// TIA Portal V15.1 export
// export: Created 2024-05-17T05:38:54.5998709Z, ExportSetting WithDefaults, DisplayName Totally Integrated Automation Portal, DisplayVersion V15.1 Update 5, DisplayName TIA Portal Openness, DisplayVersion V15.1 Update 5, DisplayName SINAMICS Startdrive Advanced, DisplayVersion V15.1, DisplayName G130, G150, S120, S150, SINAMICS MV, S210, DisplayVersion V15.1, DisplayName G110M, G120, G120C, G120D, G120P, DisplayVersion V15.1, DisplayName STEP 7 Professional, DisplayVersion V15.1 Update 5, DisplayName STEP 7 Safety, DisplayVersion V15.1, DisplayName WinCC Professional, DisplayVersion V15.1 Update 5, DisplayName SIMATIC Visualization Architect, DisplayVersion V15.1
FUNCTION "209220ZS01PNIODiag" : Void   // FC374, FBD
TITLE = 209220ZS01PNIODiag
{ S7_Optimized_Access := 'FALSE' }
AUTHOR : JS
NAME : Mot001
VERSION : 0.1
// stored: AutoNumber false, IsIECCheckEnabled false, SetENOAutomatically False, UDAEnableTagReadback false
   VAR_OUTPUT
      O_AlarmA : Bool;   // Alarm A
      O_AlarmB : Bool;   // Alarm B
      O_AlarmC : Bool;   // Alarm C
      O_AlarmD : Bool;   // Alarm D
      O_AlarmABCondition : Bool;   // Alarms resetable
      H_IAnim : Word;   // Animation bits to Icon in WinCC
   END_VAR
   VAR_TEMP   // added for the SCL form of the ladder/FBD networks
      _w1 : Bool;
   END_VAR
BEGIN

REGION Network 1: **** --------------------- ET200sp I/O --------------------- ****
END_REGION

REGION Network 2: **** 3 - Communication - Devices **** 209220AS10-JW50 - ET200sp I/O - Busnode 220AS10 - node 50
   // Profinet device don't exist - ET200sp I/O - Busnode 220AS10 - node 50
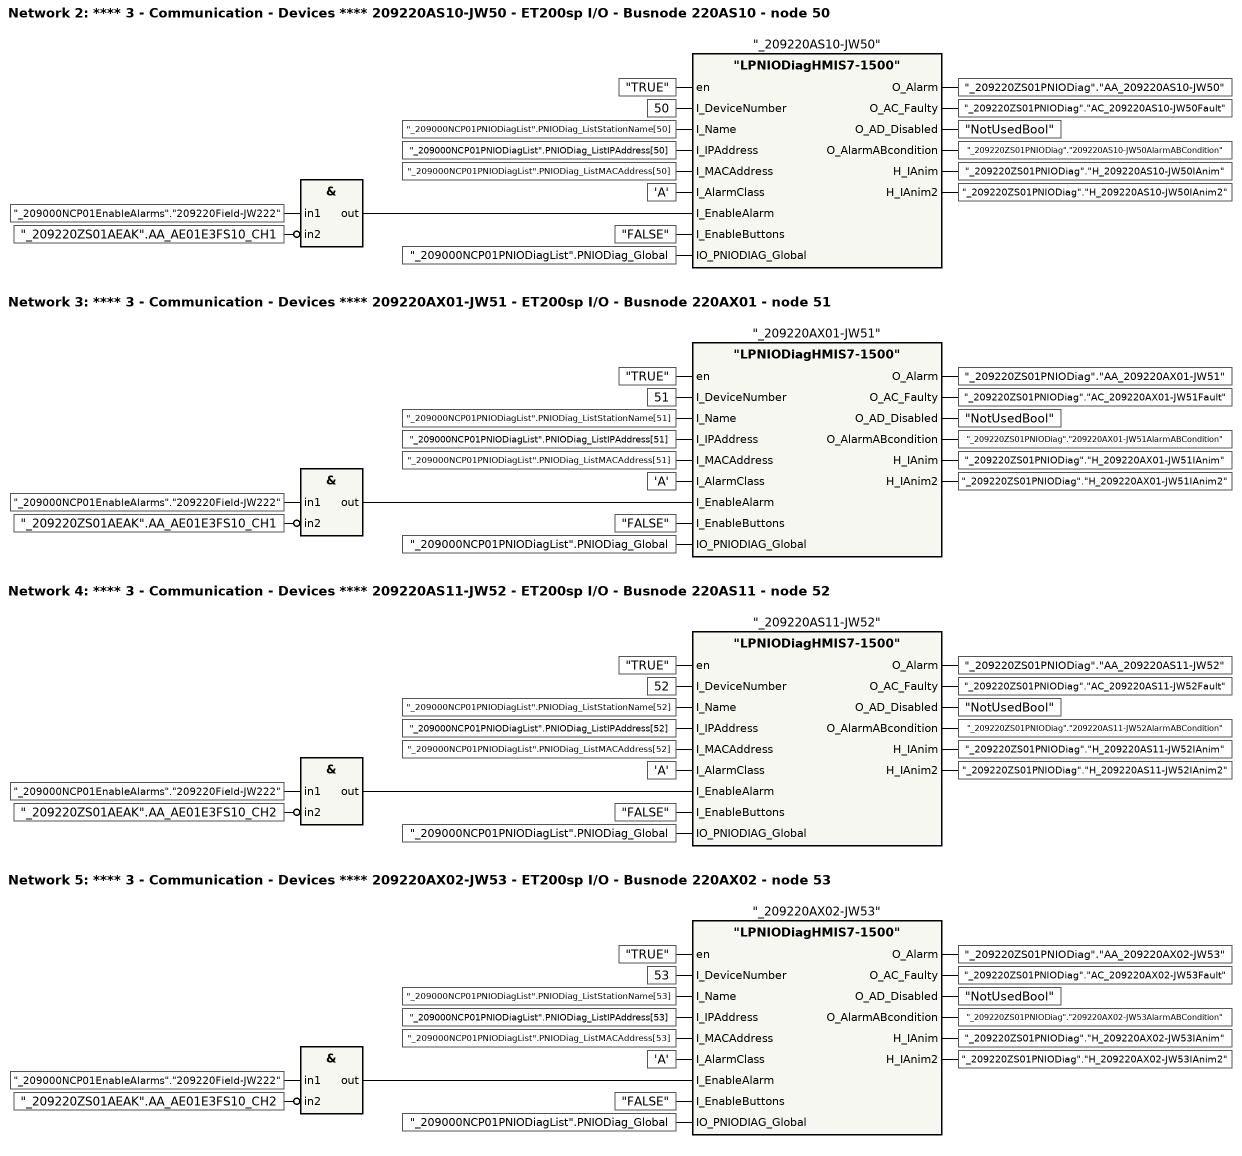
   IF "TRUE" THEN
       "_209220AS10-JW50"(I_DeviceNumber := 50,   // "LPNIODiagHMIS7-1500"
                          I_Name := "_209000NCP01PNIODiagList".PNIODiag_ListStationName[50],
                          I_IPAddress := "_209000NCP01PNIODiagList".PNIODiag_ListIPAddress[50],
                          I_MACAddress := "_209000NCP01PNIODiagList".PNIODiag_ListMACAddress[50],
                          I_AlarmClass := 'A',
                          I_EnableAlarm := "_209000NCP01EnableAlarms"."209220Field-JW222" AND NOT "_209220ZS01AEAK".AA_AE01E3FS10_CH1,
                          I_EnableButtons := "FALSE",
                          IO_PNIODIAG_Global := "_209000NCP01PNIODiagList".PNIODiag_Global,
                          O_Alarm => "_209220ZS01PNIODiag"."AA_209220AS10-JW50",
                          O_AC_Faulty => "_209220ZS01PNIODiag"."AC_209220AS10-JW50Fault",
                          O_AD_Disabled => "NotUsedBool",
                          O_AlarmABcondition => "_209220ZS01PNIODiag"."209220AS10-JW50AlarmABCondition",
                          H_IAnim => "_209220ZS01PNIODiag"."H_209220AS10-JW50IAnim",
                          H_IAnim2 => "_209220ZS01PNIODiag"."H_209220AS10-JW50IAnim2");
   END_IF;
END_REGION

REGION Network 3: **** 3 - Communication - Devices **** 209220AX01-JW51 - ET200sp I/O - Busnode 220AX01 - node 51
   // Profinet device don't exist - ET200sp I/O - Busnode 220AX01 - node 51
   IF "TRUE" THEN
       "_209220AX01-JW51"(I_DeviceNumber := 51,   // "LPNIODiagHMIS7-1500"
                          I_Name := "_209000NCP01PNIODiagList".PNIODiag_ListStationName[51],
                          I_IPAddress := "_209000NCP01PNIODiagList".PNIODiag_ListIPAddress[51],
                          I_MACAddress := "_209000NCP01PNIODiagList".PNIODiag_ListMACAddress[51],
                          I_AlarmClass := 'A',
                          I_EnableAlarm := "_209000NCP01EnableAlarms"."209220Field-JW222" AND NOT "_209220ZS01AEAK".AA_AE01E3FS10_CH1,
                          I_EnableButtons := "FALSE",
                          IO_PNIODIAG_Global := "_209000NCP01PNIODiagList".PNIODiag_Global,
                          O_Alarm => "_209220ZS01PNIODiag"."AA_209220AX01-JW51",
                          O_AC_Faulty => "_209220ZS01PNIODiag"."AC_209220AX01-JW51Fault",
                          O_AD_Disabled => "NotUsedBool",
                          O_AlarmABcondition => "_209220ZS01PNIODiag"."209220AX01-JW51AlarmABCondition",
                          H_IAnim => "_209220ZS01PNIODiag"."H_209220AX01-JW51IAnim",
                          H_IAnim2 => "_209220ZS01PNIODiag"."H_209220AX01-JW51IAnim2");
   END_IF;
END_REGION

REGION Network 4: **** 3 - Communication - Devices **** 209220AS11-JW52 - ET200sp I/O - Busnode 220AS11 - node 52
   // Profinet device don't exist - ET200sp I/O - Busnode 220AS11 - node 52
   IF "TRUE" THEN
       "_209220AS11-JW52"(I_DeviceNumber := 52,   // "LPNIODiagHMIS7-1500"
                          I_Name := "_209000NCP01PNIODiagList".PNIODiag_ListStationName[52],
                          I_IPAddress := "_209000NCP01PNIODiagList".PNIODiag_ListIPAddress[52],
                          I_MACAddress := "_209000NCP01PNIODiagList".PNIODiag_ListMACAddress[52],
                          I_AlarmClass := 'A',
                          I_EnableAlarm := "_209000NCP01EnableAlarms"."209220Field-JW222" AND NOT "_209220ZS01AEAK".AA_AE01E3FS10_CH2,
                          I_EnableButtons := "FALSE",
                          IO_PNIODIAG_Global := "_209000NCP01PNIODiagList".PNIODiag_Global,
                          O_Alarm => "_209220ZS01PNIODiag"."AA_209220AS11-JW52",
                          O_AC_Faulty => "_209220ZS01PNIODiag"."AC_209220AS11-JW52Fault",
                          O_AD_Disabled => "NotUsedBool",
                          O_AlarmABcondition => "_209220ZS01PNIODiag"."209220AS11-JW52AlarmABCondition",
                          H_IAnim => "_209220ZS01PNIODiag"."H_209220AS11-JW52IAnim",
                          H_IAnim2 => "_209220ZS01PNIODiag"."H_209220AS11-JW52IAnim2");
   END_IF;
END_REGION

REGION Network 5: **** 3 - Communication - Devices **** 209220AX02-JW53 - ET200sp I/O - Busnode 220AX02 - node 53
   // Profinet device don't exist - ET200sp I/O - Busnode 220AX02 - node 53
   IF "TRUE" THEN
       "_209220AX02-JW53"(I_DeviceNumber := 53,   // "LPNIODiagHMIS7-1500"
                          I_Name := "_209000NCP01PNIODiagList".PNIODiag_ListStationName[53],
                          I_IPAddress := "_209000NCP01PNIODiagList".PNIODiag_ListIPAddress[53],
                          I_MACAddress := "_209000NCP01PNIODiagList".PNIODiag_ListMACAddress[53],
                          I_AlarmClass := 'A',
                          I_EnableAlarm := "_209000NCP01EnableAlarms"."209220Field-JW222" AND NOT "_209220ZS01AEAK".AA_AE01E3FS10_CH2,
                          I_EnableButtons := "FALSE",
                          IO_PNIODIAG_Global := "_209000NCP01PNIODiagList".PNIODiag_Global,
                          O_Alarm => "_209220ZS01PNIODiag"."AA_209220AX02-JW53",
                          O_AC_Faulty => "_209220ZS01PNIODiag"."AC_209220AX02-JW53Fault",
                          O_AD_Disabled => "NotUsedBool",
                          O_AlarmABcondition => "_209220ZS01PNIODiag"."209220AX02-JW53AlarmABCondition",
                          H_IAnim => "_209220ZS01PNIODiag"."H_209220AX02-JW53IAnim",
                          H_IAnim2 => "_209220ZS01PNIODiag"."H_209220AX02-JW53IAnim2");
   END_IF;
END_REGION

REGION Network 6: **** 3 - Communication - Devices **** 209220AS20-JW58 - ET200sp I/O - Busnode 220AS20 - node 58
   // Profinet device don't exist - ET200sp I/O - Busnode 220AS20 - node 58
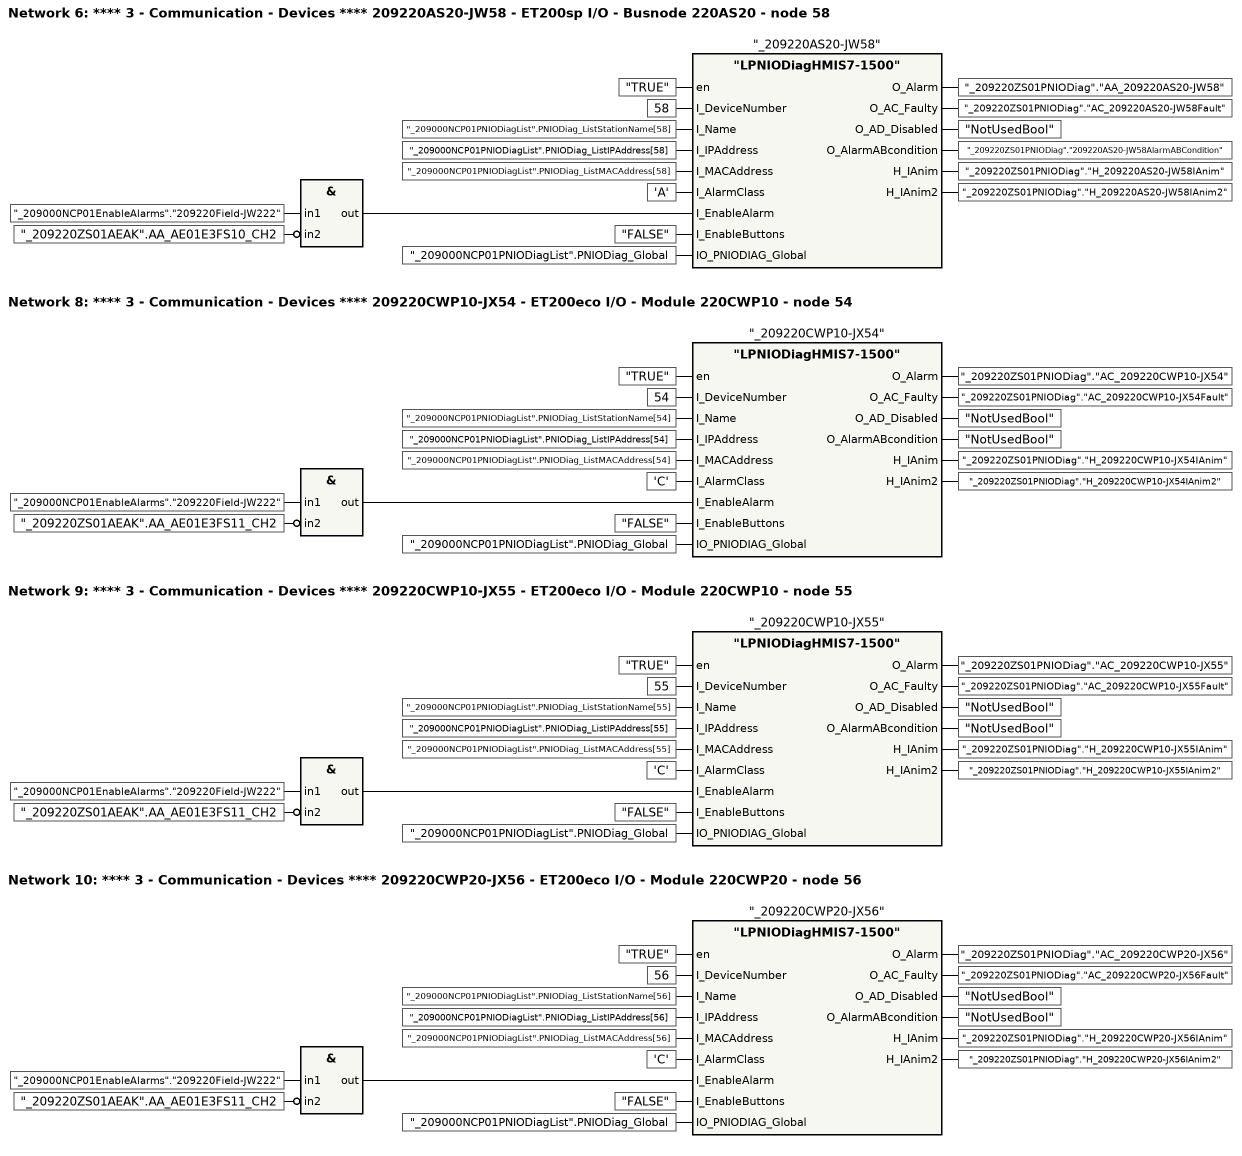
   IF "TRUE" THEN
       "_209220AS20-JW58"(I_DeviceNumber := 58,   // "LPNIODiagHMIS7-1500"
                          I_Name := "_209000NCP01PNIODiagList".PNIODiag_ListStationName[58],
                          I_IPAddress := "_209000NCP01PNIODiagList".PNIODiag_ListIPAddress[58],
                          I_MACAddress := "_209000NCP01PNIODiagList".PNIODiag_ListMACAddress[58],
                          I_AlarmClass := 'A',
                          I_EnableAlarm := "_209000NCP01EnableAlarms"."209220Field-JW222" AND NOT "_209220ZS01AEAK".AA_AE01E3FS10_CH2,
                          I_EnableButtons := "FALSE",
                          IO_PNIODIAG_Global := "_209000NCP01PNIODiagList".PNIODiag_Global,
                          O_Alarm => "_209220ZS01PNIODiag"."AA_209220AS20-JW58",
                          O_AC_Faulty => "_209220ZS01PNIODiag"."AC_209220AS20-JW58Fault",
                          O_AD_Disabled => "NotUsedBool",
                          O_AlarmABcondition => "_209220ZS01PNIODiag"."209220AS20-JW58AlarmABCondition",
                          H_IAnim => "_209220ZS01PNIODiag"."H_209220AS20-JW58IAnim",
                          H_IAnim2 => "_209220ZS01PNIODiag"."H_209220AS20-JW58IAnim2");
   END_IF;
END_REGION

REGION Network 7: **** --------------------- ET200eco I/O --------------------- ****
END_REGION

REGION Network 8: **** 3 - Communication - Devices **** 209220CWP10-JX54 - ET200eco I/O - Module 220CWP10 - node 54
   // Profinet device don't exist - ET200eco I/O - Module 220CWP10 - node 54
   IF "TRUE" THEN
       "_209220CWP10-JX54"(I_DeviceNumber := 54,   // "LPNIODiagHMIS7-1500"
                           I_Name := "_209000NCP01PNIODiagList".PNIODiag_ListStationName[54],
                           I_IPAddress := "_209000NCP01PNIODiagList".PNIODiag_ListIPAddress[54],
                           I_MACAddress := "_209000NCP01PNIODiagList".PNIODiag_ListMACAddress[54],
                           I_AlarmClass := 'C',
                           I_EnableAlarm := "_209000NCP01EnableAlarms"."209220Field-JW222" AND NOT "_209220ZS01AEAK".AA_AE01E3FS11_CH2,
                           I_EnableButtons := "FALSE",
                           IO_PNIODIAG_Global := "_209000NCP01PNIODiagList".PNIODiag_Global,
                           O_Alarm => "_209220ZS01PNIODiag"."AC_209220CWP10-JX54",
                           O_AC_Faulty => "_209220ZS01PNIODiag"."AC_209220CWP10-JX54Fault",
                           O_AD_Disabled => "NotUsedBool",
                           O_AlarmABcondition => "NotUsedBool",
                           H_IAnim => "_209220ZS01PNIODiag"."H_209220CWP10-JX54IAnim",
                           H_IAnim2 => "_209220ZS01PNIODiag"."H_209220CWP10-JX54IAnim2");
   END_IF;
END_REGION

REGION Network 9: **** 3 - Communication - Devices **** 209220CWP10-JX55 - ET200eco I/O - Module 220CWP10 - node 55
   // Profinet device don't exist - ET200eco I/O - Module 220CWP10 - node 55
   IF "TRUE" THEN
       "_209220CWP10-JX55"(I_DeviceNumber := 55,   // "LPNIODiagHMIS7-1500"
                           I_Name := "_209000NCP01PNIODiagList".PNIODiag_ListStationName[55],
                           I_IPAddress := "_209000NCP01PNIODiagList".PNIODiag_ListIPAddress[55],
                           I_MACAddress := "_209000NCP01PNIODiagList".PNIODiag_ListMACAddress[55],
                           I_AlarmClass := 'C',
                           I_EnableAlarm := "_209000NCP01EnableAlarms"."209220Field-JW222" AND NOT "_209220ZS01AEAK".AA_AE01E3FS11_CH2,
                           I_EnableButtons := "FALSE",
                           IO_PNIODIAG_Global := "_209000NCP01PNIODiagList".PNIODiag_Global,
                           O_Alarm => "_209220ZS01PNIODiag"."AC_209220CWP10-JX55",
                           O_AC_Faulty => "_209220ZS01PNIODiag"."AC_209220CWP10-JX55Fault",
                           O_AD_Disabled => "NotUsedBool",
                           O_AlarmABcondition => "NotUsedBool",
                           H_IAnim => "_209220ZS01PNIODiag"."H_209220CWP10-JX55IAnim",
                           H_IAnim2 => "_209220ZS01PNIODiag"."H_209220CWP10-JX55IAnim2");
   END_IF;
END_REGION

REGION Network 10: **** 3 - Communication - Devices **** 209220CWP20-JX56 - ET200eco I/O - Module 220CWP20 - node 56
   // Profinet device don't exist - ET200eco I/O - Module 220CWP20 - node 56
   IF "TRUE" THEN
       "_209220CWP20-JX56"(I_DeviceNumber := 56,   // "LPNIODiagHMIS7-1500"
                           I_Name := "_209000NCP01PNIODiagList".PNIODiag_ListStationName[56],
                           I_IPAddress := "_209000NCP01PNIODiagList".PNIODiag_ListIPAddress[56],
                           I_MACAddress := "_209000NCP01PNIODiagList".PNIODiag_ListMACAddress[56],
                           I_AlarmClass := 'C',
                           I_EnableAlarm := "_209000NCP01EnableAlarms"."209220Field-JW222" AND NOT "_209220ZS01AEAK".AA_AE01E3FS11_CH2,
                           I_EnableButtons := "FALSE",
                           IO_PNIODIAG_Global := "_209000NCP01PNIODiagList".PNIODiag_Global,
                           O_Alarm => "_209220ZS01PNIODiag"."AC_209220CWP20-JX56",
                           O_AC_Faulty => "_209220ZS01PNIODiag"."AC_209220CWP20-JX56Fault",
                           O_AD_Disabled => "NotUsedBool",
                           O_AlarmABcondition => "NotUsedBool",
                           H_IAnim => "_209220ZS01PNIODiag"."H_209220CWP20-JX56IAnim",
                           H_IAnim2 => "_209220ZS01PNIODiag"."H_209220CWP20-JX56IAnim2");
   END_IF;
END_REGION

REGION Network 11: **** 3 - Communication - Devices **** 209220CWP20-JX57 - ET200eco I/O - Module 220CWP20 - node 57
   // Profinet device don't exist - ET200eco I/O - Module 220CWP20 - node 57
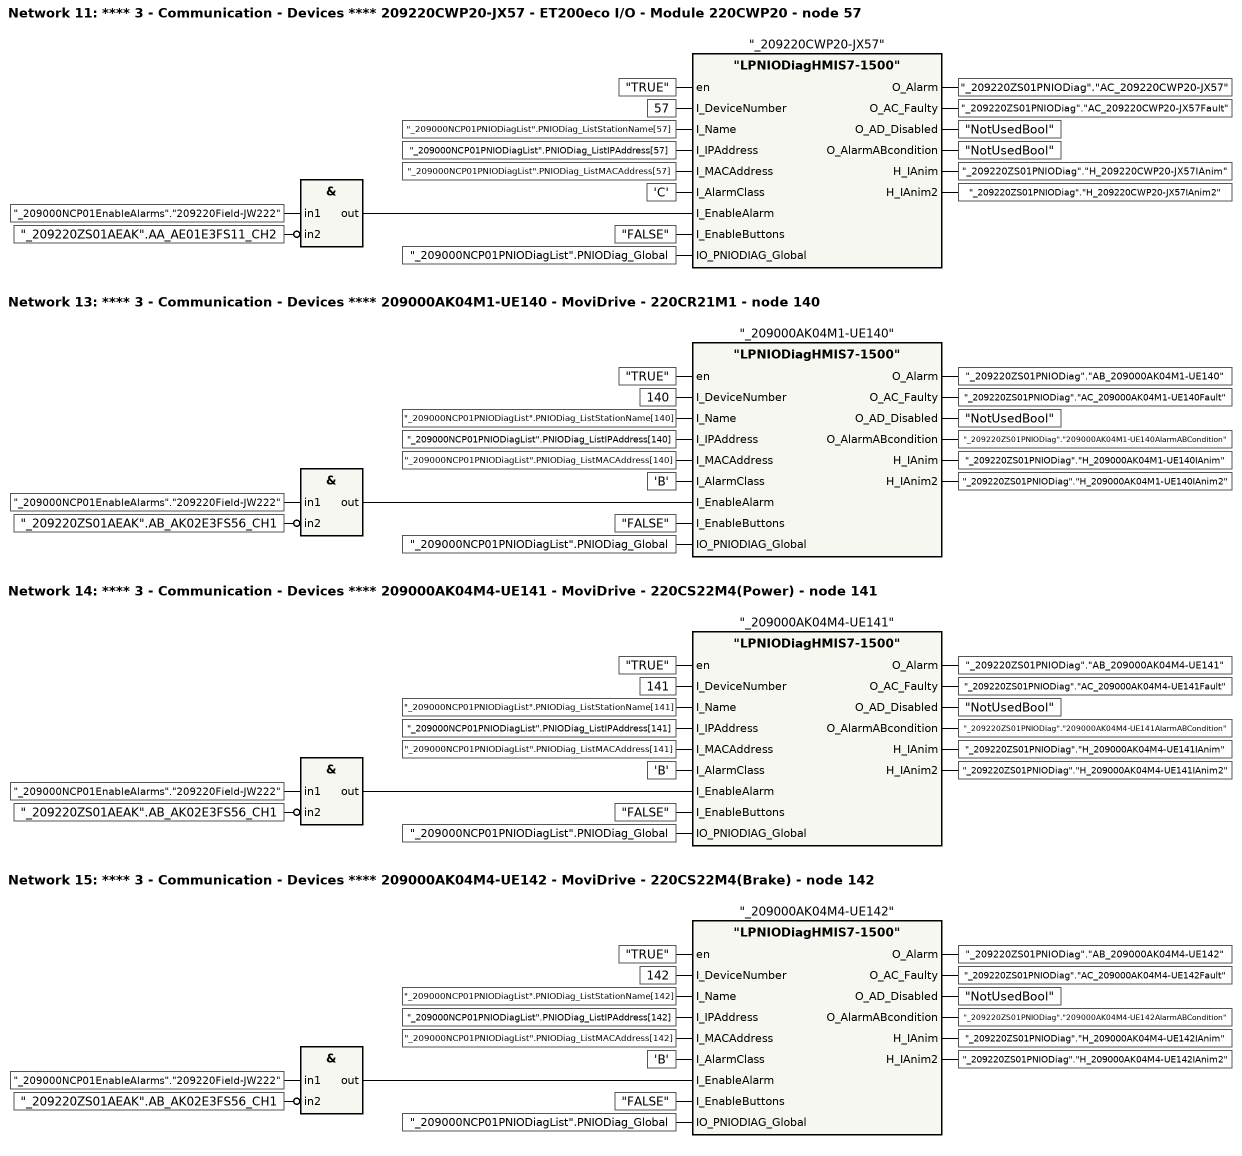
   IF "TRUE" THEN
       "_209220CWP20-JX57"(I_DeviceNumber := 57,   // "LPNIODiagHMIS7-1500"
                           I_Name := "_209000NCP01PNIODiagList".PNIODiag_ListStationName[57],
                           I_IPAddress := "_209000NCP01PNIODiagList".PNIODiag_ListIPAddress[57],
                           I_MACAddress := "_209000NCP01PNIODiagList".PNIODiag_ListMACAddress[57],
                           I_AlarmClass := 'C',
                           I_EnableAlarm := "_209000NCP01EnableAlarms"."209220Field-JW222" AND NOT "_209220ZS01AEAK".AA_AE01E3FS11_CH2,
                           I_EnableButtons := "FALSE",
                           IO_PNIODIAG_Global := "_209000NCP01PNIODiagList".PNIODiag_Global,
                           O_Alarm => "_209220ZS01PNIODiag"."AC_209220CWP20-JX57",
                           O_AC_Faulty => "_209220ZS01PNIODiag"."AC_209220CWP20-JX57Fault",
                           O_AD_Disabled => "NotUsedBool",
                           O_AlarmABcondition => "NotUsedBool",
                           H_IAnim => "_209220ZS01PNIODiag"."H_209220CWP20-JX57IAnim",
                           H_IAnim2 => "_209220ZS01PNIODiag"."H_209220CWP20-JX57IAnim2");
   END_IF;
END_REGION

REGION Network 12: **** --------------------- Drive --------------------- ****
END_REGION

REGION Network 13: **** 3 - Communication - Devices **** 209000AK04M1-UE140 - MoviDrive - 220CR21M1 - node 140
   // Profinet device don't exist - MoviDrive - 220CR21M1 - node 140
   IF "TRUE" THEN
       "_209000AK04M1-UE140"(I_DeviceNumber := 140,   // "LPNIODiagHMIS7-1500"
                             I_Name := "_209000NCP01PNIODiagList".PNIODiag_ListStationName[140],
                             I_IPAddress := "_209000NCP01PNIODiagList".PNIODiag_ListIPAddress[140],
                             I_MACAddress := "_209000NCP01PNIODiagList".PNIODiag_ListMACAddress[140],
                             I_AlarmClass := 'B',
                             I_EnableAlarm := "_209000NCP01EnableAlarms"."209220Field-JW222" AND NOT "_209220ZS01AEAK".AB_AK02E3FS56_CH1,
                             I_EnableButtons := "FALSE",
                             IO_PNIODIAG_Global := "_209000NCP01PNIODiagList".PNIODiag_Global,
                             O_Alarm => "_209220ZS01PNIODiag"."AB_209000AK04M1-UE140",
                             O_AC_Faulty => "_209220ZS01PNIODiag"."AC_209000AK04M1-UE140Fault",
                             O_AD_Disabled => "NotUsedBool",
                             O_AlarmABcondition => "_209220ZS01PNIODiag"."209000AK04M1-UE140AlarmABCondition",
                             H_IAnim => "_209220ZS01PNIODiag"."H_209000AK04M1-UE140IAnim",
                             H_IAnim2 => "_209220ZS01PNIODiag"."H_209000AK04M1-UE140IAnim2");
   END_IF;
END_REGION

REGION Network 14: **** 3 - Communication - Devices **** 209000AK04M4-UE141 - MoviDrive - 220CS22M4(Power) - node 141
   // Profinet device don't exist - MoviDrive - 220CS22M4(Power) - node 141
   IF "TRUE" THEN
       "_209000AK04M4-UE141"(I_DeviceNumber := 141,   // "LPNIODiagHMIS7-1500"
                             I_Name := "_209000NCP01PNIODiagList".PNIODiag_ListStationName[141],
                             I_IPAddress := "_209000NCP01PNIODiagList".PNIODiag_ListIPAddress[141],
                             I_MACAddress := "_209000NCP01PNIODiagList".PNIODiag_ListMACAddress[141],
                             I_AlarmClass := 'B',
                             I_EnableAlarm := "_209000NCP01EnableAlarms"."209220Field-JW222" AND NOT "_209220ZS01AEAK".AB_AK02E3FS56_CH1,
                             I_EnableButtons := "FALSE",
                             IO_PNIODIAG_Global := "_209000NCP01PNIODiagList".PNIODiag_Global,
                             O_Alarm => "_209220ZS01PNIODiag"."AB_209000AK04M4-UE141",
                             O_AC_Faulty => "_209220ZS01PNIODiag"."AC_209000AK04M4-UE141Fault",
                             O_AD_Disabled => "NotUsedBool",
                             O_AlarmABcondition => "_209220ZS01PNIODiag"."209000AK04M4-UE141AlarmABCondition",
                             H_IAnim => "_209220ZS01PNIODiag"."H_209000AK04M4-UE141IAnim",
                             H_IAnim2 => "_209220ZS01PNIODiag"."H_209000AK04M4-UE141IAnim2");
   END_IF;
END_REGION

REGION Network 15: **** 3 - Communication - Devices **** 209000AK04M4-UE142 - MoviDrive - 220CS22M4(Brake) - node 142
   // Profinet device don't exist - MoviDrive - 220CS22M4(Brake) - node 142
   IF "TRUE" THEN
       "_209000AK04M4-UE142"(I_DeviceNumber := 142,   // "LPNIODiagHMIS7-1500"
                             I_Name := "_209000NCP01PNIODiagList".PNIODiag_ListStationName[142],
                             I_IPAddress := "_209000NCP01PNIODiagList".PNIODiag_ListIPAddress[142],
                             I_MACAddress := "_209000NCP01PNIODiagList".PNIODiag_ListMACAddress[142],
                             I_AlarmClass := 'B',
                             I_EnableAlarm := "_209000NCP01EnableAlarms"."209220Field-JW222" AND NOT "_209220ZS01AEAK".AB_AK02E3FS56_CH1,
                             I_EnableButtons := "FALSE",
                             IO_PNIODIAG_Global := "_209000NCP01PNIODiagList".PNIODiag_Global,
                             O_Alarm => "_209220ZS01PNIODiag"."AB_209000AK04M4-UE142",
                             O_AC_Faulty => "_209220ZS01PNIODiag"."AC_209000AK04M4-UE142Fault",
                             O_AD_Disabled => "NotUsedBool",
                             O_AlarmABcondition => "_209220ZS01PNIODiag"."209000AK04M4-UE142AlarmABCondition",
                             H_IAnim => "_209220ZS01PNIODiag"."H_209000AK04M4-UE142IAnim",
                             H_IAnim2 => "_209220ZS01PNIODiag"."H_209000AK04M4-UE142IAnim2");
   END_IF;
END_REGION

REGION Network 16: **** 3 - Communication - Devices **** 209000AK04M1-UE143 - MoviDrive - 220CR23M1 - node 143
   // Profinet device don't exist - MoviDrive - 220CR23M1 - node 143
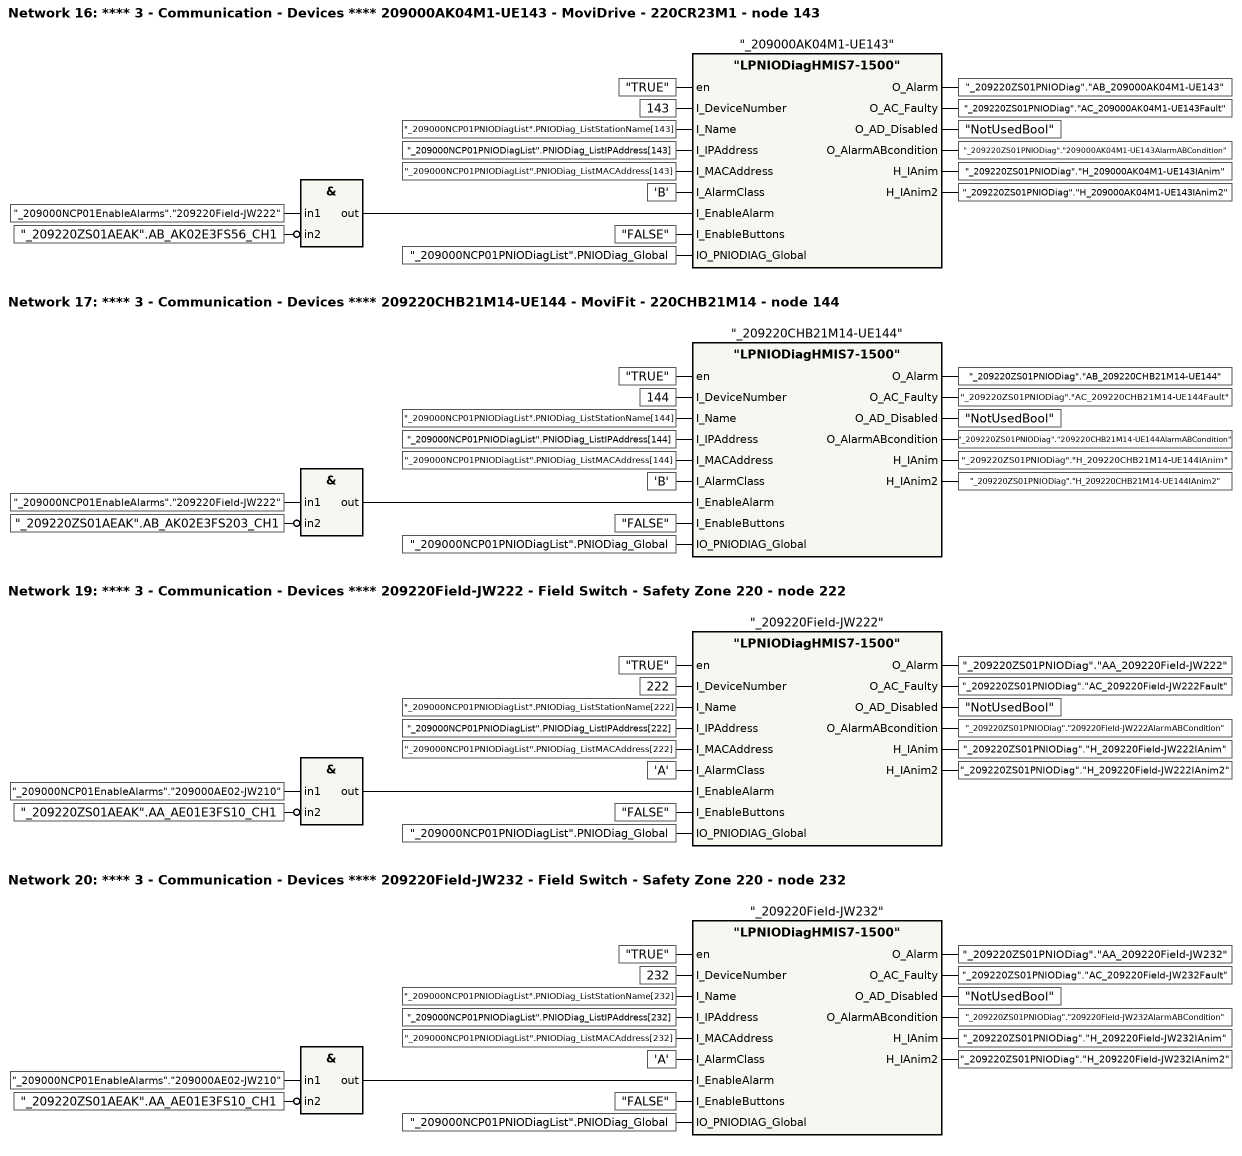
   IF "TRUE" THEN
       "_209000AK04M1-UE143"(I_DeviceNumber := 143,   // "LPNIODiagHMIS7-1500"
                             I_Name := "_209000NCP01PNIODiagList".PNIODiag_ListStationName[143],
                             I_IPAddress := "_209000NCP01PNIODiagList".PNIODiag_ListIPAddress[143],
                             I_MACAddress := "_209000NCP01PNIODiagList".PNIODiag_ListMACAddress[143],
                             I_AlarmClass := 'B',
                             I_EnableAlarm := "_209000NCP01EnableAlarms"."209220Field-JW222" AND NOT "_209220ZS01AEAK".AB_AK02E3FS56_CH1,
                             I_EnableButtons := "FALSE",
                             IO_PNIODIAG_Global := "_209000NCP01PNIODiagList".PNIODiag_Global,
                             O_Alarm => "_209220ZS01PNIODiag"."AB_209000AK04M1-UE143",
                             O_AC_Faulty => "_209220ZS01PNIODiag"."AC_209000AK04M1-UE143Fault",
                             O_AD_Disabled => "NotUsedBool",
                             O_AlarmABcondition => "_209220ZS01PNIODiag"."209000AK04M1-UE143AlarmABCondition",
                             H_IAnim => "_209220ZS01PNIODiag"."H_209000AK04M1-UE143IAnim",
                             H_IAnim2 => "_209220ZS01PNIODiag"."H_209000AK04M1-UE143IAnim2");
   END_IF;
END_REGION

REGION Network 17: **** 3 - Communication - Devices **** 209220CHB21M14-UE144 - MoviFit - 220CHB21M14 - node 144
   // Profinet device don't exist - MoviFit - 220CHB21M14 - node 144
   IF "TRUE" THEN
       "_209220CHB21M14-UE144"(I_DeviceNumber := 144,   // "LPNIODiagHMIS7-1500"
                               I_Name := "_209000NCP01PNIODiagList".PNIODiag_ListStationName[144],
                               I_IPAddress := "_209000NCP01PNIODiagList".PNIODiag_ListIPAddress[144],
                               I_MACAddress := "_209000NCP01PNIODiagList".PNIODiag_ListMACAddress[144],
                               I_AlarmClass := 'B',
                               I_EnableAlarm := "_209000NCP01EnableAlarms"."209220Field-JW222" AND NOT "_209220ZS01AEAK".AB_AK02E3FS203_CH1,
                               I_EnableButtons := "FALSE",
                               IO_PNIODIAG_Global := "_209000NCP01PNIODiagList".PNIODiag_Global,
                               O_Alarm => "_209220ZS01PNIODiag"."AB_209220CHB21M14-UE144",
                               O_AC_Faulty => "_209220ZS01PNIODiag"."AC_209220CHB21M14-UE144Fault",
                               O_AD_Disabled => "NotUsedBool",
                               O_AlarmABcondition => "_209220ZS01PNIODiag"."209220CHB21M14-UE144AlarmABCondition",
                               H_IAnim => "_209220ZS01PNIODiag"."H_209220CHB21M14-UE144IAnim",
                               H_IAnim2 => "_209220ZS01PNIODiag"."H_209220CHB21M14-UE144IAnim2");
   END_IF;
END_REGION

REGION Network 18: **** --------------------- Field Switch --------------------- ****
END_REGION

REGION Network 19: **** 3 - Communication - Devices **** 209220Field-JW222 - Field Switch - Safety Zone 220 - node 222
   // Profinet device don't exist - Field Switch - Safety Zone 220 - node 222
   IF "TRUE" THEN
       "_209220Field-JW222"(I_DeviceNumber := 222,   // "LPNIODiagHMIS7-1500"
                            I_Name := "_209000NCP01PNIODiagList".PNIODiag_ListStationName[222],
                            I_IPAddress := "_209000NCP01PNIODiagList".PNIODiag_ListIPAddress[222],
                            I_MACAddress := "_209000NCP01PNIODiagList".PNIODiag_ListMACAddress[222],
                            I_AlarmClass := 'A',
                            I_EnableAlarm := "_209000NCP01EnableAlarms"."209000AE02-JW210" AND NOT "_209220ZS01AEAK".AA_AE01E3FS10_CH1,
                            I_EnableButtons := "FALSE",
                            IO_PNIODIAG_Global := "_209000NCP01PNIODiagList".PNIODiag_Global,
                            O_Alarm => "_209220ZS01PNIODiag"."AA_209220Field-JW222",
                            O_AC_Faulty => "_209220ZS01PNIODiag"."AC_209220Field-JW222Fault",
                            O_AD_Disabled => "NotUsedBool",
                            O_AlarmABcondition => "_209220ZS01PNIODiag"."209220Field-JW222AlarmABCondition",
                            H_IAnim => "_209220ZS01PNIODiag"."H_209220Field-JW222IAnim",
                            H_IAnim2 => "_209220ZS01PNIODiag"."H_209220Field-JW222IAnim2");
   END_IF;
END_REGION

REGION Network 20: **** 3 - Communication - Devices **** 209220Field-JW232 - Field Switch - Safety Zone 220 - node 232
   // Profinet device don't exist - Field Switch - Safety Zone 220 - node 232
   IF "TRUE" THEN
       "_209220Field-JW232"(I_DeviceNumber := 232,   // "LPNIODiagHMIS7-1500"
                            I_Name := "_209000NCP01PNIODiagList".PNIODiag_ListStationName[232],
                            I_IPAddress := "_209000NCP01PNIODiagList".PNIODiag_ListIPAddress[232],
                            I_MACAddress := "_209000NCP01PNIODiagList".PNIODiag_ListMACAddress[232],
                            I_AlarmClass := 'A',
                            I_EnableAlarm := "_209000NCP01EnableAlarms"."209000AE02-JW210" AND NOT "_209220ZS01AEAK".AA_AE01E3FS10_CH1,
                            I_EnableButtons := "FALSE",
                            IO_PNIODIAG_Global := "_209000NCP01PNIODiagList".PNIODiag_Global,
                            O_Alarm => "_209220ZS01PNIODiag"."AA_209220Field-JW232",
                            O_AC_Faulty => "_209220ZS01PNIODiag"."AC_209220Field-JW232Fault",
                            O_AD_Disabled => "NotUsedBool",
                            O_AlarmABcondition => "_209220ZS01PNIODiag"."209220Field-JW232AlarmABCondition",
                            H_IAnim => "_209220ZS01PNIODiag"."H_209220Field-JW232IAnim",
                            H_IAnim2 => "_209220ZS01PNIODiag"."H_209220Field-JW232IAnim2");
   END_IF;
END_REGION

REGION Network 21: **** -------------------------------------------------- ****
END_REGION

REGION Network 22: **** 4.6 - Machine Status - Indications **** Icon animation
   // Icon animation
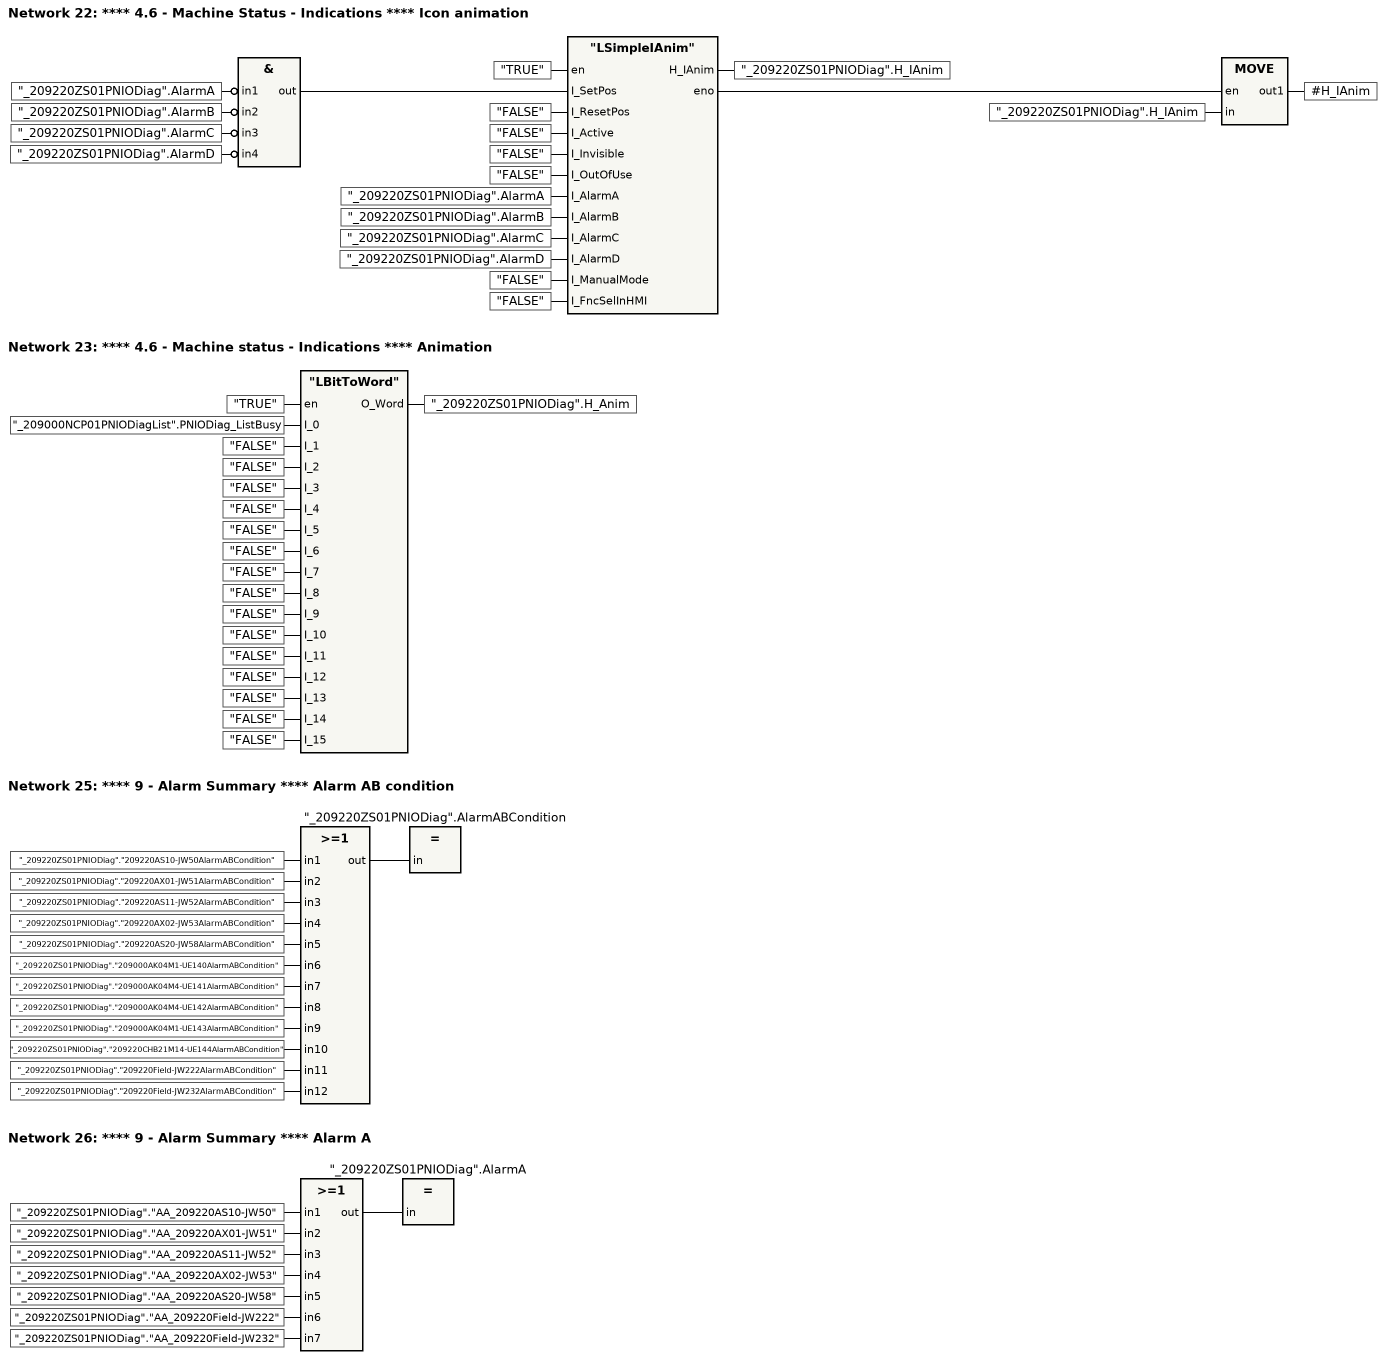
   "LSimpleIAnim"(EN := "TRUE",
                  I_SetPos := NOT "_209220ZS01PNIODiag".AlarmA AND NOT "_209220ZS01PNIODiag".AlarmB AND NOT "_209220ZS01PNIODiag".AlarmC AND NOT "_209220ZS01PNIODiag".AlarmD,
                  I_ResetPos := "FALSE",
                  I_Active := "FALSE",
                  I_Invisible := "FALSE",
                  I_OutOfUse := "FALSE",
                  I_AlarmA := "_209220ZS01PNIODiag".AlarmA,
                  I_AlarmB := "_209220ZS01PNIODiag".AlarmB,
                  I_AlarmC := "_209220ZS01PNIODiag".AlarmC,
                  I_AlarmD := "_209220ZS01PNIODiag".AlarmD,
                  I_ManualMode := "FALSE",
                  I_FncSelInHMI := "FALSE",
                  H_IAnim => "_209220ZS01PNIODiag".H_IAnim,
                  ENO => #_w1);
   IF #_w1 THEN #H_IAnim := "_209220ZS01PNIODiag".H_IAnim; END_IF;
END_REGION

REGION Network 23: **** 4.6 - Machine status - Indications **** Animation
   // Animation
   IF "TRUE" THEN
       "LBitToWord"(I_0 := "_209000NCP01PNIODiagList".PNIODiag_ListBusy,
                    I_1 := "FALSE",
                    I_2 := "FALSE",
                    I_3 := "FALSE",
                    I_4 := "FALSE",
                    I_5 := "FALSE",
                    I_6 := "FALSE",
                    I_7 := "FALSE",
                    I_8 := "FALSE",
                    I_9 := "FALSE",
                    I_10 := "FALSE",
                    I_11 := "FALSE",
                    I_12 := "FALSE",
                    I_13 := "FALSE",
                    I_14 := "FALSE",
                    I_15 := "FALSE",
                    O_Word => "_209220ZS01PNIODiag".H_Anim);
   END_IF;
END_REGION

NETWORK
TITLE = **** 4.6 - Machine Status - Indications **** Animation DB number
// DB number
      OPN   "_209220ZS01PNIODiag";
      L     DBNO;
      T     "_209220ZS01PNIODiag".H_DBnr;

REGION Network 25: **** 9 - Alarm Summary **** Alarm AB condition
   // Summary of Alarm AB condition
   "_209220ZS01PNIODiag".AlarmABCondition := "_209220ZS01PNIODiag"."209220AS10-JW50AlarmABCondition" OR "_209220ZS01PNIODiag"."209220AX01-JW51AlarmABCondition" OR "_209220ZS01PNIODiag"."209220AS11-JW52AlarmABCondition" OR "_209220ZS01PNIODiag"."209220AX02-JW53AlarmABCondition" OR "_209220ZS01PNIODiag"."209220AS20-JW58AlarmABCondition" OR "_209220ZS01PNIODiag"."209000AK04M1-UE140AlarmABCondition" OR "_209220ZS01PNIODiag"."209000AK04M4-UE141AlarmABCondition" OR "_209220ZS01PNIODiag"."209000AK04M4-UE142AlarmABCondition" OR "_209220ZS01PNIODiag"."209000AK04M1-UE143AlarmABCondition" OR "_209220ZS01PNIODiag"."209220CHB21M14-UE144AlarmABCondition" OR "_209220ZS01PNIODiag"."209220Field-JW222AlarmABCondition" OR "_209220ZS01PNIODiag"."209220Field-JW232AlarmABCondition";
END_REGION

REGION Network 26: **** 9 - Alarm Summary **** Alarm A
   // Summary of alarms A
   "_209220ZS01PNIODiag".AlarmA := "_209220ZS01PNIODiag"."AA_209220AS10-JW50" OR "_209220ZS01PNIODiag"."AA_209220AX01-JW51" OR "_209220ZS01PNIODiag"."AA_209220AS11-JW52" OR "_209220ZS01PNIODiag"."AA_209220AX02-JW53" OR "_209220ZS01PNIODiag"."AA_209220AS20-JW58" OR "_209220ZS01PNIODiag"."AA_209220Field-JW222" OR "_209220ZS01PNIODiag"."AA_209220Field-JW232";
END_REGION

REGION Network 27: **** 9 - Alarm Summary **** Alarm B
   // Summary of alarms B
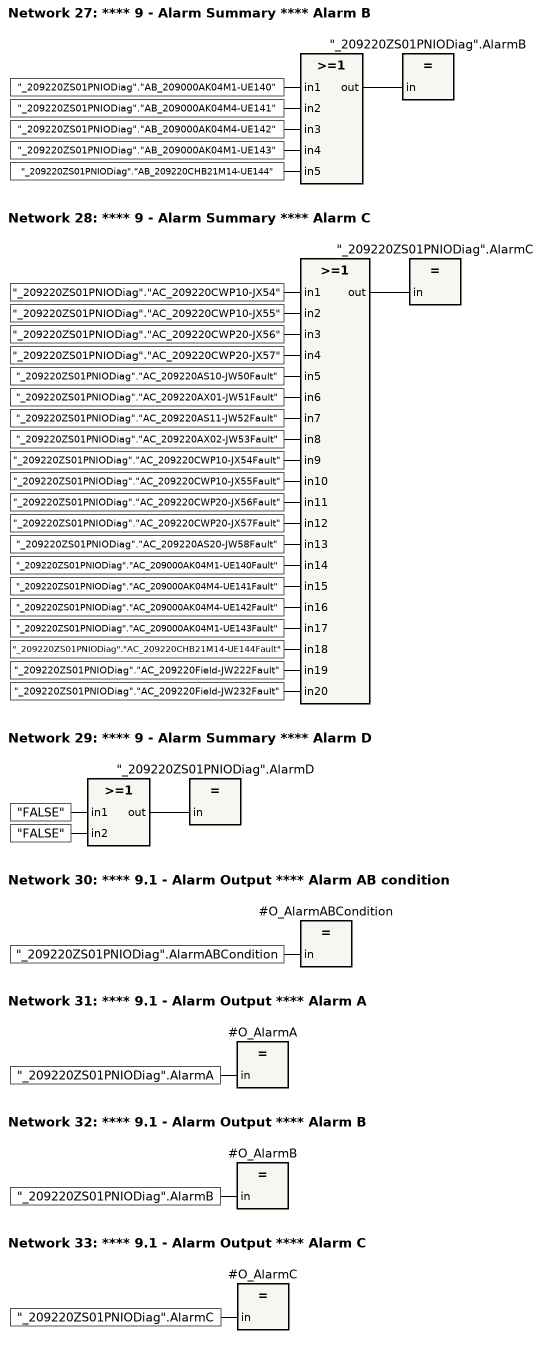
   "_209220ZS01PNIODiag".AlarmB := "_209220ZS01PNIODiag"."AB_209000AK04M1-UE140" OR "_209220ZS01PNIODiag"."AB_209000AK04M4-UE141" OR "_209220ZS01PNIODiag"."AB_209000AK04M4-UE142" OR "_209220ZS01PNIODiag"."AB_209000AK04M1-UE143" OR "_209220ZS01PNIODiag"."AB_209220CHB21M14-UE144";
END_REGION

REGION Network 28: **** 9 - Alarm Summary **** Alarm C
   // Summary of alarms C
   "_209220ZS01PNIODiag".AlarmC := "_209220ZS01PNIODiag"."AC_209220CWP10-JX54" OR "_209220ZS01PNIODiag"."AC_209220CWP10-JX55" OR "_209220ZS01PNIODiag"."AC_209220CWP20-JX56" OR "_209220ZS01PNIODiag"."AC_209220CWP20-JX57" OR "_209220ZS01PNIODiag"."AC_209220AS10-JW50Fault" OR "_209220ZS01PNIODiag"."AC_209220AX01-JW51Fault" OR "_209220ZS01PNIODiag"."AC_209220AS11-JW52Fault" OR "_209220ZS01PNIODiag"."AC_209220AX02-JW53Fault" OR "_209220ZS01PNIODiag"."AC_209220CWP10-JX54Fault" OR "_209220ZS01PNIODiag"."AC_209220CWP10-JX55Fault" OR "_209220ZS01PNIODiag"."AC_209220CWP20-JX56Fault" OR "_209220ZS01PNIODiag"."AC_209220CWP20-JX57Fault" OR "_209220ZS01PNIODiag"."AC_209220AS20-JW58Fault" OR "_209220ZS01PNIODiag"."AC_209000AK04M1-UE140Fault" OR "_209220ZS01PNIODiag"."AC_209000AK04M4-UE141Fault" OR "_209220ZS01PNIODiag"."AC_209000AK04M4-UE142Fault" OR "_209220ZS01PNIODiag"."AC_209000AK04M1-UE143Fault" OR "_209220ZS01PNIODiag"."AC_209220CHB21M14-UE144Fault" OR "_209220ZS01PNIODiag"."AC_209220Field-JW222Fault" OR "_209220ZS01PNIODiag"."AC_209220Field-JW232Fault";
END_REGION

REGION Network 29: **** 9 - Alarm Summary **** Alarm D
   // Summary of alarms D
   "_209220ZS01PNIODiag".AlarmD := "FALSE" OR "FALSE";
END_REGION

REGION Network 30: **** 9.1 - Alarm Output **** Alarm AB condition
   // Alarm AB condition
   #O_AlarmABCondition := "_209220ZS01PNIODiag".AlarmABCondition;
END_REGION

REGION Network 31: **** 9.1 - Alarm Output **** Alarm A
   // Output Alarm A
   #O_AlarmA := "_209220ZS01PNIODiag".AlarmA;
END_REGION

REGION Network 32: **** 9.1 - Alarm Output **** Alarm B
   // Output Alarm B
   #O_AlarmB := "_209220ZS01PNIODiag".AlarmB;
END_REGION

REGION Network 33: **** 9.1 - Alarm Output **** Alarm C
   // Output Alarm A
   #O_AlarmC := "_209220ZS01PNIODiag".AlarmC;
END_REGION

REGION Network 34: **** 9.1 - Alarm Output **** Alarm D
   // Output Alarm D
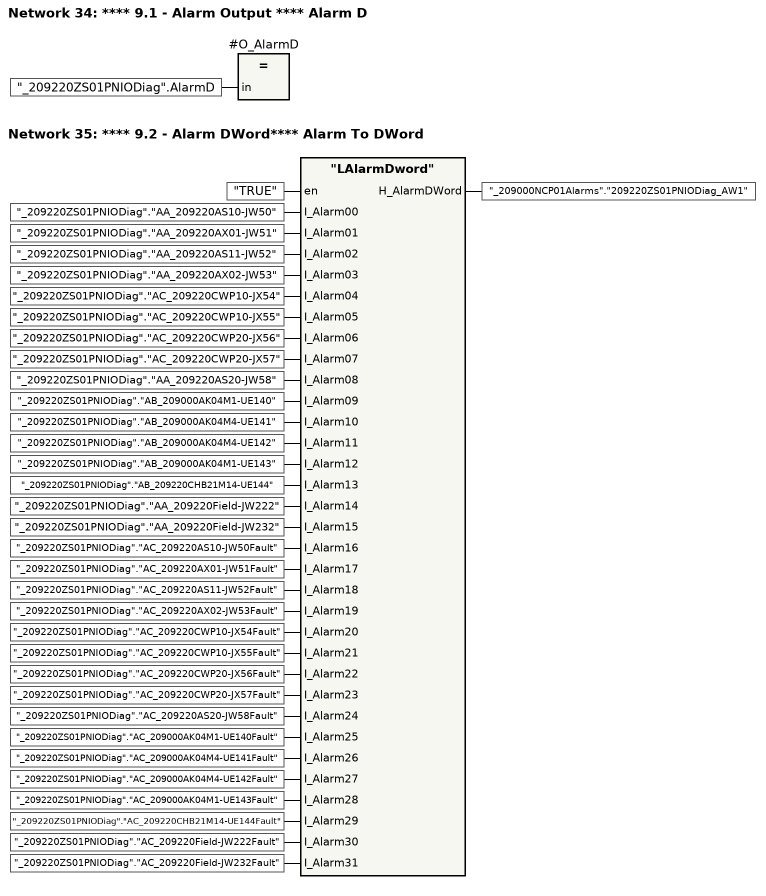
   #O_AlarmD := "_209220ZS01PNIODiag".AlarmD;
END_REGION

REGION Network 35: **** 9.2 - Alarm DWord**** Alarm To DWord
   // Alarm Word
   IF "TRUE" THEN
       "LAlarmDword"(I_Alarm00 := "_209220ZS01PNIODiag"."AA_209220AS10-JW50",
                     I_Alarm01 := "_209220ZS01PNIODiag"."AA_209220AX01-JW51",
                     I_Alarm02 := "_209220ZS01PNIODiag"."AA_209220AS11-JW52",
                     I_Alarm03 := "_209220ZS01PNIODiag"."AA_209220AX02-JW53",
                     I_Alarm04 := "_209220ZS01PNIODiag"."AC_209220CWP10-JX54",
                     I_Alarm05 := "_209220ZS01PNIODiag"."AC_209220CWP10-JX55",
                     I_Alarm06 := "_209220ZS01PNIODiag"."AC_209220CWP20-JX56",
                     I_Alarm07 := "_209220ZS01PNIODiag"."AC_209220CWP20-JX57",
                     I_Alarm08 := "_209220ZS01PNIODiag"."AA_209220AS20-JW58",
                     I_Alarm09 := "_209220ZS01PNIODiag"."AB_209000AK04M1-UE140",
                     I_Alarm10 := "_209220ZS01PNIODiag"."AB_209000AK04M4-UE141",
                     I_Alarm11 := "_209220ZS01PNIODiag"."AB_209000AK04M4-UE142",
                     I_Alarm12 := "_209220ZS01PNIODiag"."AB_209000AK04M1-UE143",
                     I_Alarm13 := "_209220ZS01PNIODiag"."AB_209220CHB21M14-UE144",
                     I_Alarm14 := "_209220ZS01PNIODiag"."AA_209220Field-JW222",
                     I_Alarm15 := "_209220ZS01PNIODiag"."AA_209220Field-JW232",
                     I_Alarm16 := "_209220ZS01PNIODiag"."AC_209220AS10-JW50Fault",
                     I_Alarm17 := "_209220ZS01PNIODiag"."AC_209220AX01-JW51Fault",
                     I_Alarm18 := "_209220ZS01PNIODiag"."AC_209220AS11-JW52Fault",
                     I_Alarm19 := "_209220ZS01PNIODiag"."AC_209220AX02-JW53Fault",
                     I_Alarm20 := "_209220ZS01PNIODiag"."AC_209220CWP10-JX54Fault",
                     I_Alarm21 := "_209220ZS01PNIODiag"."AC_209220CWP10-JX55Fault",
                     I_Alarm22 := "_209220ZS01PNIODiag"."AC_209220CWP20-JX56Fault",
                     I_Alarm23 := "_209220ZS01PNIODiag"."AC_209220CWP20-JX57Fault",
                     I_Alarm24 := "_209220ZS01PNIODiag"."AC_209220AS20-JW58Fault",
                     I_Alarm25 := "_209220ZS01PNIODiag"."AC_209000AK04M1-UE140Fault",
                     I_Alarm26 := "_209220ZS01PNIODiag"."AC_209000AK04M4-UE141Fault",
                     I_Alarm27 := "_209220ZS01PNIODiag"."AC_209000AK04M4-UE142Fault",
                     I_Alarm28 := "_209220ZS01PNIODiag"."AC_209000AK04M1-UE143Fault",
                     I_Alarm29 := "_209220ZS01PNIODiag"."AC_209220CHB21M14-UE144Fault",
                     I_Alarm30 := "_209220ZS01PNIODiag"."AC_209220Field-JW222Fault",
                     I_Alarm31 := "_209220ZS01PNIODiag"."AC_209220Field-JW232Fault",
                     H_AlarmDWord => "_209000NCP01Alarms"."209220ZS01PNIODiag_AW1");
   END_IF;
END_REGION
END_FUNCTION
